FUNCTION_BLOCK EL4014
VAR
	_io : EL4xx4_Data;
	{attribute addProperty Name "WcState"}
	_wcState : WcStateBase;
	{attribute addProperty Name "Info data"}
	_infoData : InfoDataAds;
END_VAR

PROPERTY IO : REFERENCE TO EL4xx4_Data
GET
IO REF= _io;
END_GET
END_PROPERTY

PROPERTY WcState : REFERENCE TO WcStateBase
GET
WcState REF= _wcState;
END_GET
END_PROPERTY

END_FUNCTION_BLOCK

(* stored: Version 1.1.0.1, ProductVersion 3.1.4024.9
   POU EL4014: Id {6f2210a2-b74f-09c0-2b2a-3bb0d687acbb}, SpecialFunc None
   Property IO: Id {704aaa5e-c903-0076-07db-9d84746169eb}
   Get Get: Id {9b11a1ed-d3f0-0517-1f8f-a7b3551e5d12}
   Property WcState: Id {10e50837-82d9-007a-1c5c-934cd4a7c2b9}
   Get Get: Id {effe78ac-44cd-03b3-38f9-4a527a538bc5} *)
